// TIA Portal project "MiniFluffy" (V17)

(* hardware
DEVICE "S7-1200 station_1"  S7-1200 Station
   slot 0: "Rack_0"  S7-1200 Rack  Rack  V1.0
   slot 1: "PLC_1"  CPU 1212FC DC/DC/RLY  6ES7 212-1HF40-0XB0  V4.5
   slot 2: "DI 16/DQ 16x24VDC_1"  6ES7 223-1BL32-0XB0  V2.0
   slot 3: "DQ 16x24VDC_1"  SM 1222 DQ16 x 24VDC  6ES7 222-1BH32-0XB0  V2.0
*)

// ===== PLC "PLC_1"  CPU 1212FC DC/DC/RLY =====

VAR_GLOBAL   // PLC tag table "Default tag table"
   "System_OK" AT %M100.0 : Bool;
   "TU1_Busy" AT %M100.1 : Bool;
   "TU2_Busy" AT %M100.2 : Bool;
   "Error_Code_01" AT %M100.7 : Bool;
   "Channel1_Active" AT %M101.0 : Bool;
   "Channel2_Active" AT %M101.1 : Bool;
   "Channel3_Active" AT %M101.2 : Bool;
   "Channel4_Active" AT %M101.3 : Bool;
   "PO1_Busy" AT %M101.4 : Bool;
   "PO2_Busy" AT %M101.5 : Bool;
   "PO3_Busy" AT %M101.6 : Bool;
   "TU1_Reset" AT %M102.1 : Bool;
   "TU2_Reset" AT %M102.2 : Bool;
   "PO1_Reset" AT %M102.3 : Bool;
   "PO2_Reset" AT %M102.4 : Bool;
   "PO3_Reset" AT %M102.5 : Bool;
   "SO1_1_Reset" AT %M102.6 : Bool;
   "SO1_2_Reset" AT %M102.7 : Bool;
   "SO1_3_Reset" AT %M103.0 : Bool;
   "SO1_4_Reset" AT %M103.1 : Bool;
   "SO1_5_Reset" AT %M103.2 : Bool;
   "SO2_1_Reset" AT %M103.3 : Bool;
   "SO2_2_Reset" AT %M103.4 : Bool;
   "SO2_3_Reset" AT %M103.5 : Bool;
   "SO2_4_Reset" AT %M103.6 : Bool;
   "SO2_5_Reset" AT %M103.7 : Bool;
   "SO1_1_Error" AT %M104.0 : Bool;
   "SO1_2_Error" AT %M104.1 : Bool;
   "SO1_3_Error" AT %M104.2 : Bool;
   "SO1_4_Error" AT %M104.3 : Bool;
   "SO1_5_Error" AT %M104.4 : Bool;
   "SO2_1_Error" AT %M104.5 : Bool;
   "SO2_2_Error" AT %M104.6 : Bool;
   "SO2_3_Error" AT %M104.7 : Bool;
   "SO2_4_Error" AT %M105.0 : Bool;
   "SO2_5_Error" AT %M105.1 : Bool;
   "Clock_1Hz" AT %M0.5 : Bool;
   "FirstScan" AT %M1.0 : Bool;
   "Station1_Mode" AT %M105.2 : Bool;
   "Station2_Mode" AT %M105.3 : Bool;
   "Station3_Mode" AT %M105.4 : Bool;
   "PO1_Time" AT %MD110 : Time;
   "PO2_Time" AT %MD115 : Time;
   "PO3_Time" AT %MD120 : Time;
   "PO1_Manual_Ack" AT %M105.5 : Bool;
   "PO2_Manual_Ack" AT %M105.6 : Bool;
   "PO3_Manual_Ack" AT %M105.7 : Bool;
   "PO1_Positioned" AT %M106.0 : Bool;
   "PO2_Positioned" AT %M106.1 : Bool;
   "PO3_Positioned" AT %M106.2 : Bool;
   "First_Init" AT %M106.3 : Bool;
   "EME_Active" AT %M106.5 : Bool;
END_VAR

VAR_GLOBAL   // PLC tag table "I/O list"
   "Magnetic1_1" AT %I8.0 : Bool;   // Magnetic proximity sensor conveyor belt 1 position 1
   "Magnetic1_2" AT %I8.1 : Bool;   // Magnetic proximity sensor conveyor belt 1 position 2
   "Magnetic1_3" AT %I8.2 : Bool;   // Magnetic proximity sensor conveyor belt 1 position 3
   "Magnetic1_4" AT %I8.3 : Bool;   // Magnetic proximity sensor conveyor belt 1 position 4
   "Magnetic1_5" AT %I8.4 : Bool;   // Magnetic proximity sensor conveyor belt 1 position 5
   "Magnetic2_1" AT %I8.5 : Bool;   // Magnetic proximity sensor conveyor belt 2 position 1
   "Magnetic2_2" AT %I8.6 : Bool;   // Magnetic proximity sensor conveyor belt 2 position 2
   "Magnetic2_3" AT %I8.7 : Bool;   // Magnetic proximity sensor conveyor belt 2 position 3
   "Magnetic2_4" AT %I9.0 : Bool;   // Magnetic proximity sensor conveyor belt 2 position 4
   "Magnetic2_5" AT %I9.1 : Bool;   // Magnetic proximity sensor conveyor belt 2 position 5
   "TU1_IndBuf" AT %I9.2 : Bool;   // Inductive sensor product carrier transfer unit 1, buffer sensor
   "TU2_IndBuf" AT %I9.3 : Bool;   // Inductive sensor product carrier transfer unit 2, buffer sensor
   "System_Safe" AT %I0.0 : Bool;   // Output Safety relay acknowledge system is safe
   "PO1_LinAct_Down" AT %Q8.0 : Bool;   // Linear Actuator product carrier transfer unit 1 move up
   "PO1_LinAct_Up" AT %Q8.1 : Bool;   // Linear Actuator product carrier transfer unit 1 move down
   "PO2_LinAct_Down" AT %Q8.2 : Bool;   // Linear Actuator product carrier transfer unit 2 move up
   "PO2_LinAct_Up" AT %Q8.3 : Bool;   // Linear Actuator product carrier transfer unit 2 move down
   "PO3_LinAct_Down" AT %Q8.4 : Bool;   // Linear Actuator positioner 1 move up
   "PO3_LinAct_Up" AT %Q8.5 : Bool;   // Linear Actuator positioner 1 move down
   "TU1_LinAct_Down" AT %Q8.6 : Bool;   // Linear Actuator positioner 2 move up
   "TU1_LinAct_Up" AT %Q8.7 : Bool;   // Linear Actuator positioner 2 move down
   "TU2_LinAct_Down" AT %Q9.0 : Bool;   // Linear Actuator positioner 3 move up
   "TU2_LinAct_Up" AT %Q9.1 : Bool;   // Linear Actuator positioner 3 move down
   "Solenoid_SP1_1" AT %Q12.0 : Bool;   // Activate the solenoid for Stopper 1 on conveyor 1
   "Solenoid_SP1_2" AT %Q12.1 : Bool;   // Activate the solenoid for Stopper 2 on conveyor 1
   "Solenoid_SP1_3" AT %Q12.2 : Bool;   // Activate the solenoid for Stopper 3 on conveyor 1
   "Solenoid_SP1_4" AT %Q12.3 : Bool;   // Activate the solenoid for Stopper 4 on conveyor 1
   "Solenoid_SP1_5" AT %Q12.4 : Bool;   // Activate the solenoid for Stopper 5 on conveyor 1
   "Solenoid_SP2_1" AT %Q12.5 : Bool;   // Activate the solenoid for Stopper 1 on conveyor 2
   "Solenoid_SP2_2" AT %Q12.6 : Bool;   // Activate the solenoid for Stopper 2 on conveyor 2
   "Solenoid_SP2_3" AT %Q12.7 : Bool;   // Activate the solenoid for Stopper 3 on conveyor 2
   "Solenoid_SP2_4" AT %Q13.0 : Bool;   // Activate the solenoid for Stopper 4 on conveyor 2
   "Solenoid_SP2_5" AT %Q13.1 : Bool;   // Activate the solenoid for Stopper 5 on conveyor 2
   "AC_Motor_RLY" AT %Q9.5 : Bool;   // Power up/Power down the AC Motor Relay
   "TU1_DC_Motor" AT %Q9.6 : Bool;   // Power up/Power down the product carrier transfer unit 1 Relay
   "TU2_DC_Motor" AT %Q9.7 : Bool;   // Power up/Power down the product carrier transfer unit 2 Relay
   "Eme_Stop_1" AT %I0.1 : Bool;   // Emergency stop 1, 2nd NC signal
   "Eme_Stop_2" AT %I0.2 : Bool;   // Emergency stop 2, 2nd NC signal
   "Reset_LED" AT %Q9.4 : Bool;   // Reset LED for the Pilz safety relay
   "Red_LED" AT %Q0.2 : Bool;   // Red LED for the signal tower
   "Green_LED" AT %Q0.0 : Bool;   // Green LED for the signal tower
   "Yellow_LED" AT %Q0.1 : Bool;   // Yellow LED for the signal tower
   "12 V DC ok" AT %I0.3 : Bool;   // 12 V DC power supply is OK
   "Communication_SelectivyModule" AT %I0.4 : Bool;
END_VAR

DATA_BLOCK "Main_Safety_RTG1_DB"   // DB1, F_DB
{ S7_Optimized_Access := 'TRUE' }
NAME : FUSI
VERSION : 0.1
// stored: InstanceOfName Main_Safety_RTG1
"Main_Safety_RTG1"
BEGIN
END_DATA_BLOCK

DATA_BLOCK "tranfer_station_DB"   // DB2
{ S7_Optimized_Access := 'TRUE' }
VERSION : 0.1
// stored: InstanceOfName tranfer_station
"tranfer_station"
BEGIN
END_DATA_BLOCK

FUNCTION_BLOCK "Main_Safety_RTG1"   // FB1, F_FBD
{ S7_Optimized_Access := 'TRUE' }
BEGIN
END_FUNCTION_BLOCK

FUNCTION_BLOCK "po_lift_stop"   // FB2, LAD
{ S7_Optimized_Access := 'TRUE' }
VERSION : 0.1
   VAR_INPUT
      next_station_free : Bool;
      magnetic : Bool;
   END_VAR
   VAR_OUTPUT
      solenoid_out : Bool;
      lift_up : Bool;
      lift_down : Bool;
   END_VAR
   VAR
      raise_po_timer : TP_TIME;
      lower_po_timer : TON_TIME;
   END_VAR
   VAR_TEMP
      StationDone : Bool;
   END_VAR
BEGIN

REGION Network 1 (SCL)
   IF #magnetic THEN
       #raise_po_timer.TP(IN:= NOT #lower_po_timer.Q,
                              PT:= T#15s);
           #lift_up := #raise_po_timer.Q;
           #lift_down := NOT #raise_po_timer.Q;
           #solenoid_out := NOT #raise_po_timer.Q AND #next_station_free;
           IF NOT #raise_po_timer.Q AND #next_station_free THEN
               #lower_po_timer.TON(IN := TRUE,
                                 PT := T#2s);
             IF #lower_po_timer.Q THEN
                #raise_po_timer.IN := FALSE;
                #raise_po_timer.IN := FALSE;
            END_IF;
        END_IF;
    END_IF;
END_REGION
END_FUNCTION_BLOCK

FUNCTION_BLOCK "tranfer_station"   // FB3, SCL
{ S7_Optimized_Access := 'TRUE' }
VERSION : 0.1
   VAR_INPUT
      magnetic_start : Bool;
      magnetic_end : Bool;
      induction_mid : Bool;
   END_VAR
   VAR_OUTPUT
      lift_up : Bool;
      lift_down : Bool;
      conveyor : Bool;
   END_VAR
   VAR
      station_active : Bool;
      done_lifting_timer : TON_TIME;
      delay_conveyor : TON_TIME;
      start_lifting : Bool;
   END_VAR
BEGIN
   #done_lifting_timer(IN :=#start_lifting, PT := T#2s);
   IF #magnetic_start THEN
       #station_active := TRUE;
       #done_lifting_timer.IN := FALSE;
       #delay_conveyor.IN := FALSE;
   END_IF;
   IF #station_active THEN
       #lift_up := TRUE;
       #lift_down := FALSE;
       #start_lifting := TRUE;
       IF #done_lifting_timer.Q THEN
           #start_lifting := FALSE;
           #conveyor := TRUE;
       END_IF;
       IF #magnetic_end THEN
           #delay_conveyor(IN:=TRUE,
                           PT:=T#3s);
           IF #delay_conveyor.Q THEN
               #lift_up := FALSE;
               #lift_down := TRUE;
               #conveyor := FALSE;
               #station_active := FALSE;
           END_IF;
       END_IF;
   END_IF;
END_FUNCTION_BLOCK

ORGANIZATION_BLOCK "Main"   // OB1, LAD, ProgramCycle
TITLE = "Main Program Sweep (Cycle)"
{ S7_Optimized_Access := 'TRUE' }
VERSION : 0.1
   VAR_INPUT
      Initial_Call : Bool;   // Initial call of this OB
      Remanence : Bool;   // =True, if remanent data are available
   END_VAR
BEGIN

REGION Network 1: Check System Safety
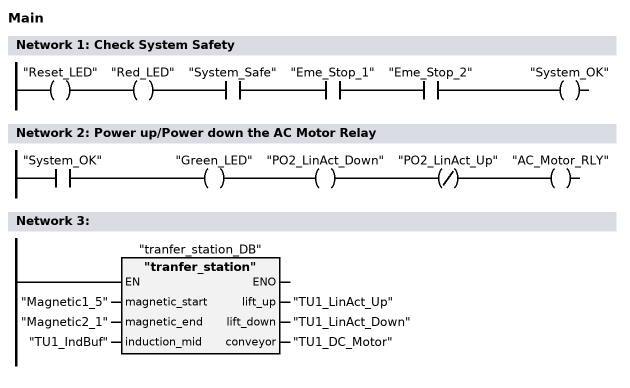
   RUNG wire#powerrail
      Coil( "Reset_LED" )
      Coil( "Red_LED" )
      Contact( "System_Safe" )
      Contact( "Eme_Stop_1" )
      Contact( "Eme_Stop_2" )
      Coil( "System_OK" )
   END_RUNG
   // the same network as SCL:
   "Reset_LED" := TRUE;
   "Red_LED" := TRUE;
   "System_OK" := "System_Safe" AND "Eme_Stop_1" AND "Eme_Stop_2";
END_REGION

REGION Network 2: Power up/Power down the AC Motor Relay
   RUNG wire#powerrail
      Contact( "System_OK" )
      Coil( "Green_LED" )
      Coil( "PO2_LinAct_Down" )
      I_Coil( "PO2_LinAct_Up" )
      Coil( "AC_Motor_RLY" )
   END_RUNG
   // the same network as SCL:
   "Green_LED" := "System_OK";
   "PO2_LinAct_Down" := "System_OK";
   "PO2_LinAct_Up" := NOT "System_OK";
   "AC_Motor_RLY" := "System_OK";
END_REGION

REGION Network 3
   RUNG wire#powerrail
      "tranfer_station_DB"(magnetic_start := "Magnetic1_5", magnetic_end := "Magnetic2_1", induction_mid := "TU1_IndBuf", lift_up => "TU1_LinAct_Up", lift_down => "TU1_LinAct_Down", conveyor => "TU1_DC_Motor")
   END_RUNG
   // the same network as SCL:
   "tranfer_station_DB"(magnetic_start := "Magnetic1_5",   // "tranfer_station"
                        magnetic_end := "Magnetic2_1",
                        induction_mid := "TU1_IndBuf",
                        lift_up => "TU1_LinAct_Up",
                        lift_down => "TU1_LinAct_Down",
                        conveyor => "TU1_DC_Motor");
END_REGION
END_ORGANIZATION_BLOCK